ABB RAPID module: Module1.mod

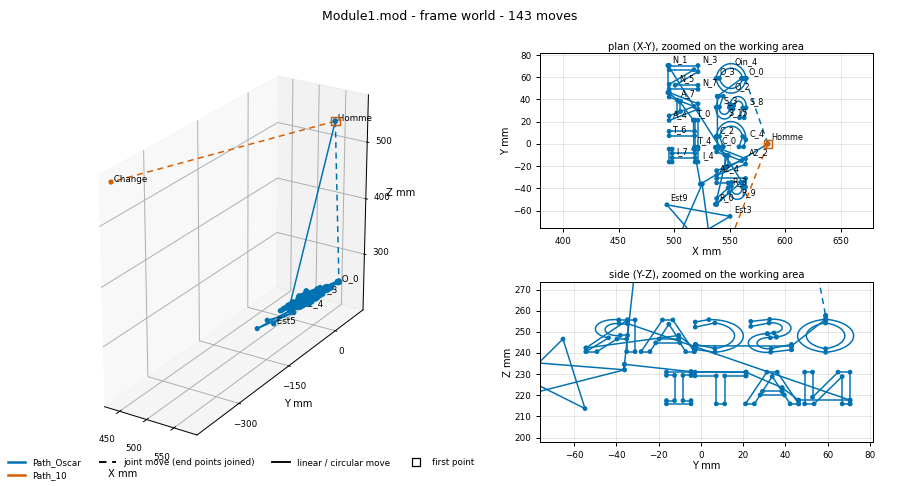
[picture p0: tool path of Module1.mod in frame world, 143 of 143 moves have a stored position in this frame; points joined in program order, loops and branches not executed]
MODULE Module1
    TASK PERS tooldata Marcador:=[TRUE,[[59.777,0,124.777],[0.923879533,0,0.382683432,0]],[0.105,[17.009,0,56.388],[1,0,0,0],0,0,0]];
    TASK PERS wobjdata Pastel:=[FALSE,TRUE,"",[[480,-5.202,208],[0.258819045,0,0.965925826,0]],[[-17.44,75.771,0.905],[0,0,1,0]]];
    CONST robtarget N_1:=[[0,0,2],[0,0,1,0],[-1,1,-2,0],[9E+09,9E+09,9E+09,9E+09,9E+09,9E+09]];
    CONST robtarget N_2:=[[0,0,0],[0,0,1,0],[-1,1,-2,0],[9E+09,9E+09,9E+09,9E+09,9E+09,9E+09]];
    CONST robtarget N_3:=[[30,0,0],[0,0,1,0],[-1,1,-2,0],[9E+09,9E+09,9E+09,9E+09,9E+09,9E+09]];
    CONST robtarget N_4:=[[30,-5.664,0],[0,0,1,0],[-1,1,-2,0],[9E+09,9E+09,9E+09,9E+09,9E+09,9E+09]];
    CONST robtarget N_5:=[[6.248,-17.747,0],[0,0,1,0],[-1,1,-2,0],[9E+09,9E+09,9E+09,9E+09,9E+09,9E+09]];
    CONST robtarget N_6:=[[30,-17.747,0],[0,0,1,0],[-1,1,-2,0],[9E+09,9E+09,9E+09,9E+09,9E+09,9E+09]];
    CONST robtarget N_7:=[[30,-21.467,0],[0,0,1,0],[-1,1,-2,0],[9E+09,9E+09,9E+09,9E+09,9E+09,9E+09]];
    CONST robtarget N_8:=[[-0.000025404,-21.467,0.000044001],[0,0,1,0],[-1,1,-2,0],[9E+09,9E+09,9E+09,9E+09,9E+09,9E+09]];
    CONST robtarget N_9:=[[-0.000025404,-16.993,0.000044001],[0,0,1,0],[-1,1,-2,0],[9E+09,9E+09,9E+09,9E+09,9E+09,9E+09]];
    CONST robtarget N_10:=[[25.867,-3.719,0],[0,0,1,0],[-1,1,-2,0],[9E+09,9E+09,9E+09,9E+09,9E+09,9E+09]];
    CONST robtarget N_11:=[[0,-3.719,0],[0,0,1,0],[-1,1,-2,0],[9E+09,9E+09,9E+09,9E+09,9E+09,9E+09]];
    CONST robtarget N_1_2:=[[0,0,2],[0,0,1,0],[-1,1,-2,0],[9E+09,9E+09,9E+09,9E+09,9E+09,9E+09]];
    CONST robtarget A_0:=[[0,-24.311,2],[0,0,1,0],[-1,1,-2,0],[9E+09,9E+09,9E+09,9E+09,9E+09,9E+09]];
    CONST robtarget A_1:=[[0,-24.311,0],[0,0,1,0],[-1,1,-2,0],[9E+09,9E+09,9E+09,9E+09,9E+09,9E+09]];
    CONST robtarget A_2:=[[30,-34.425,0],[0,0,1,0],[-1,1,-2,0],[9E+09,9E+09,9E+09,9E+09,9E+09,9E+09]];
    CONST robtarget A_3:=[[30,-39.335,0],[0,0,1,0],[-1,1,-2,0],[9E+09,9E+09,9E+09,9E+09,9E+09,9E+09]];
    CONST robtarget A_4:=[[0,-49.449,0],[0,0,1,0],[-1,1,-2,0],[9E+09,9E+09,9E+09,9E+09,9E+09,9E+09]];
    CONST robtarget A_5:=[[0,-45.243,0],[0,0,1,0],[-1,1,-2,0],[9E+09,9E+09,9E+09,9E+09,9E+09,9E+09]];
    CONST robtarget A_6:=[[8.388,-42.52,0],[0,0,1,0],[-1,1,-2,0],[9E+09,9E+09,9E+09,9E+09,9E+09,9E+09]];
    CONST robtarget A_7:=[[8.388,-31.07,0],[0,0,1,0],[-1,1,-2,0],[9E+09,9E+09,9E+09,9E+09,9E+09,9E+09]];
    CONST robtarget A_8:=[[0,-28.347,0],[0,0,1,0],[-1,1,-2,0],[9E+09,9E+09,9E+09,9E+09,9E+09,9E+09]];
    CONST robtarget A_1_2:=[[0,-24.311,0],[0,0,1,0],[-1,1,-2,0],[9E+09,9E+09,9E+09,9E+09,9E+09,9E+09]];
    CONST robtarget A_0_2:=[[0,-24.311,2],[0,0,1,0],[-1,1,-2,0],[9E+09,9E+09,9E+09,9E+09,9E+09,9E+09]];
    CONST robtarget A_in0:=[[11.791,-32.164,2],[0,0,1,0],[-1,1,-2,0],[9E+09,9E+09,9E+09,9E+09,9E+09,9E+09]];
    CONST robtarget A_in1:=[[11.791,-32.164,0],[0,0,1,0],[-1,1,-2,0],[9E+09,9E+09,9E+09,9E+09,9E+09,9E+09]];
    CONST robtarget A_in2:=[[25.916,-36.783,0],[0,0,1,0],[-1,1,-2,0],[9E+09,9E+09,9E+09,9E+09,9E+09,9E+09]];
    CONST robtarget A_in3:=[[11.791,-41.426,0],[0,0,1,0],[-1,1,-2,0],[9E+09,9E+09,9E+09,9E+09,9E+09,9E+09]];
    CONST robtarget A_in1_2:=[[11.791,-32.164,0],[0,0,1,0],[-1,1,-2,0],[9E+09,9E+09,9E+09,9E+09,9E+09,9E+09]];
    CONST robtarget A_in0_2:=[[11.791,-32.164,2],[0,0,1,0],[-1,1,-2,0],[9E+09,9E+09,9E+09,9E+09,9E+09,9E+09]];
    CONST robtarget I_0:=[[26.937,-75.219,2],[0,0,1,0],[-1,1,-2,0],[9E+09,9E+09,9E+09,9E+09,9E+09,9E+09]];
    CONST robtarget I_2:=[[26.937,-75.219,0],[0,0,1,0],[-1,1,-2,0],[9E+09,9E+09,9E+09,9E+09,9E+09,9E+09]];
    CONST robtarget I_3:=[[30,-75.219,0],[0,0,1,0],[-1,1,-2,0],[9E+09,9E+09,9E+09,9E+09,9E+09,9E+09]];
    CONST robtarget I_4:=[[30,-86.839,0],[0,0,1,0],[-1,1,-2,0],[9E+09,9E+09,9E+09,9E+09,9E+09,9E+09]];
    CONST robtarget I_5:=[[26.937,-86.839,0],[0,0,1,0],[-1,1,-2,0],[9E+09,9E+09,9E+09,9E+09,9E+09,9E+09]];
    CONST robtarget I_6:=[[26.937,-83.023,0],[0,0,1,0],[-1,1,-2,0],[9E+09,9E+09,9E+09,9E+09,9E+09,9E+09]];
    CONST robtarget I_7:=[[3.063,-83.023,0],[0,0,1,0],[-1,1,-2,0],[9E+09,9E+09,9E+09,9E+09,9E+09,9E+09]];
    CONST robtarget I_8:=[[3.063,-86.839,0],[0,0,1,0],[-1,1,-2,0],[9E+09,9E+09,9E+09,9E+09,9E+09,9E+09]];
    CONST robtarget I_9:=[[0,-86.839,0],[0,0,1,0],[-1,1,-2,0],[9E+09,9E+09,9E+09,9E+09,9E+09,9E+09]];
    CONST robtarget I_10:=[[0,-75.219,0],[0,0,1,0],[-1,1,-2,0],[9E+09,9E+09,9E+09,9E+09,9E+09,9E+09]];
    CONST robtarget I_11:=[[3.063,-75.219,0],[0,0,1,0],[-1,1,-2,0],[9E+09,9E+09,9E+09,9E+09,9E+09,9E+09]];
    CONST robtarget I_12:=[[3.063,-79.036,0],[0,0,1,0],[-1,1,-2,0],[9E+09,9E+09,9E+09,9E+09,9E+09,9E+09]];
    CONST robtarget I_13:=[[26.937,-79.036,0],[0,0,1,0],[-1,1,-2,0],[9E+09,9E+09,9E+09,9E+09,9E+09,9E+09]];
    CONST robtarget I_2_2:=[[26.937,-75.219,0],[0,0,1,0],[-1,1,-2,0],[9E+09,9E+09,9E+09,9E+09,9E+09,9E+09]];
    CONST robtarget I_0_2:=[[26.937,-75.219,2],[0,0,1,0],[-1,1,-2,0],[9E+09,9E+09,9E+09,9E+09,9E+09,9E+09]];
    CONST robtarget T_0:=[[26.451,-49.23,2],[0,0,1,0],[-1,1,-2,0],[9E+09,9E+09,9E+09,9E+09,9E+09,9E+09]];
    CONST robtarget T_1:=[[26.451,-49.23,0],[0,0,1,0],[-1,1,-2,0],[9E+09,9E+09,9E+09,9E+09,9E+09,9E+09]];
    CONST robtarget T_2:=[[30,-49.23,0],[0,0,1,0],[-1,1,-2,0],[9E+09,9E+09,9E+09,9E+09,9E+09,9E+09]];
    CONST robtarget T_3:=[[30,-73.347,0],[0,0,1,0],[-1,1,-2,0],[9E+09,9E+09,9E+09,9E+09,9E+09,9E+09]];
    CONST robtarget T_4:=[[26.451,-73.347,0],[0,0,1,0],[-1,1,-2,0],[9E+09,9E+09,9E+09,9E+09,9E+09,9E+09]];
    CONST robtarget T_5:=[[26.451,-63.282,0],[0,0,1,0],[-1,1,-2,0],[9E+09,9E+09,9E+09,9E+09,9E+09,9E+09]];
    CONST robtarget T_6:=[[0,-63.282,0],[0,0,1,0],[-1,1,-2,0],[9E+09,9E+09,9E+09,9E+09,9E+09,9E+09]];
    CONST robtarget T_7:=[[0,-59.295,0],[0,0,1,0],[-1,1,-2,0],[9E+09,9E+09,9E+09,9E+09,9E+09,9E+09]];
    CONST robtarget T_8:=[[26.451,-59.295,0],[0,0,1,0],[-1,1,-2,0],[9E+09,9E+09,9E+09,9E+09,9E+09,9E+09]];
    CONST robtarget T_1_2:=[[26.451,-49.23,0],[0,0,1,0],[-1,1,-2,0],[9E+09,9E+09,9E+09,9E+09,9E+09,9E+09]];
    CONST robtarget T_0_2:=[[26.451,-49.23,2],[0,0,1,0],[-1,1,-2,0],[9E+09,9E+09,9E+09,9E+09,9E+09,9E+09]];
    CONST robtarget A2_0:=[[49.394,-73.711,2],[0,0,1,0],[-1,1,-2,0],[9E+09,9E+09,9E+09,9E+09,9E+09,9E+09]];
    CONST robtarget A2_1:=[[49.394,-73.711,0],[0,0,1,0],[-1,1,-2,0],[9E+09,9E+09,9E+09,9E+09,9E+09,9E+09]];
    CONST robtarget A2_2:=[[79.394,-83.825,0],[0,0,1,0],[-1,1,-2,0],[9E+09,9E+09,9E+09,9E+09,9E+09,9E+09]];
    CONST robtarget A2_3:=[[79.394,-88.736,0],[0,0,1,0],[-1,1,-2,0],[9E+09,9E+09,9E+09,9E+09,9E+09,9E+09]];
    CONST robtarget A2_4:=[[49.394,-98.849,0],[0,0,1,0],[-1,1,-2,0],[9E+09,9E+09,9E+09,9E+09,9E+09,9E+09]];
    CONST robtarget A2_5:=[[49.394,-94.643,0],[0,0,1,0],[-1,1,-2,0],[9E+09,9E+09,9E+09,9E+09,9E+09,9E+09]];
    CONST robtarget A2_6:=[[57.782,-91.92,0],[0,0,1,0],[-1,1,-2,0],[9E+09,9E+09,9E+09,9E+09,9E+09,9E+09]];
    CONST robtarget A2_7:=[[57.782,-80.47,0],[0,0,1,0],[-1,1,-2,0],[9E+09,9E+09,9E+09,9E+09,9E+09,9E+09]];
    CONST robtarget A2_8:=[[49.394,-77.747,0],[0,0,1,0],[-1,1,-2,0],[9E+09,9E+09,9E+09,9E+09,9E+09,9E+09]];
    CONST robtarget A2_1_2:=[[49.394,-73.711,0],[0,0,1,0],[-1,1,-2,0],[9E+09,9E+09,9E+09,9E+09,9E+09,9E+09]];
    CONST robtarget A2_0_2:=[[49.394,-73.711,2],[0,0,1,0],[-1,1,-2,0],[9E+09,9E+09,9E+09,9E+09,9E+09,9E+09]];
    CONST robtarget C_0:=[[51.437,-73.225,2],[0,0,1,0],[-1,1,-2,0],[9E+09,9E+09,9E+09,9E+09,9E+09,9E+09]];
    CONST robtarget C_1:=[[51.437,-73.225,0],[0,0,1,0],[-1,1,-2,0],[9E+09,9E+09,9E+09,9E+09,9E+09,9E+09]];
    CONST robtarget C_2:=[[48.86,-63.89,0],[0,0,1,0],[-1,1,-2,0],[9E+09,9E+09,9E+09,9E+09,9E+09,9E+09]];
    CONST robtarget C_3:=[[64.37,-50.47,0],[0,0,1,0],[-1,1,-2,0],[9E+09,9E+09,9E+09,9E+09,9E+09,9E+09]];
    CONST robtarget C_4:=[[79.71,-66.795,0],[0,0,1,0],[-1,1,-2,0],[9E+09,9E+09,9E+09,9E+09,9E+09,9E+09]];
    CONST robtarget C_5:=[[77.401,-73.225,0],[0,0,1,0],[-1,1,-2,0],[9E+09,9E+09,9E+09,9E+09,9E+09,9E+09]];
    CONST robtarget C_6:=[[72.587,-73.225,0],[0,0,1,0],[-1,1,-2,0],[9E+09,9E+09,9E+09,9E+09,9E+09,9E+09]];
    CONST robtarget C_7:=[[76.526,-63.938,0],[0,0,1,0],[-1,1,-2,0],[9E+09,9E+09,9E+09,9E+09,9E+09,9E+09]];
    CONST robtarget C_8:=[[64.37,-54.627,0],[0,0,1,0],[-1,1,-2,0],[9E+09,9E+09,9E+09,9E+09,9E+09,9E+09]];
    CONST robtarget C_9:=[[52.312,-63.938,0],[0,0,1,0],[-1,1,-2,0],[9E+09,9E+09,9E+09,9E+09,9E+09,9E+09]];
    CONST robtarget C_10:=[[56.202,-72.933,0],[0,0,1,0],[-1,1,-2,0],[9E+09,9E+09,9E+09,9E+09,9E+09,9E+09]];
    CONST robtarget C_11:=[[56.202,-73.225,0],[0,0,1,0],[-1,1,-2,0],[9E+09,9E+09,9E+09,9E+09,9E+09,9E+09]];
    CONST robtarget C_1_2:=[[51.437,-73.225,0],[0,0,1,0],[-1,1,-2,0],[9E+09,9E+09,9E+09,9E+09,9E+09,9E+09]];
    CONST robtarget S_0:=[[51.193,-27.715,2],[0,0,1,0],[-1,1,-2,0],[9E+09,9E+09,9E+09,9E+09,9E+09,9E+09]];
    CONST robtarget S_1:=[[51.193,-27.715,0],[0,0,1,0],[-1,1,-2,0],[9E+09,9E+09,9E+09,9E+09,9E+09,9E+09]];
    CONST robtarget S_2:=[[56.202,-27.715,0],[0,0,1,0],[-1,1,-2,0],[9E+09,9E+09,9E+09,9E+09,9E+09,9E+09]];
    CONST robtarget S_3:=[[52.312,-37.269,0],[0,0,1,0],[-1,1,-2,0],[9E+09,9E+09,9E+09,9E+09,9E+09,9E+09]];
    CONST robtarget S_4:=[[57.32,-43.954,0],[0,0,1,0],[-1,1,-2,0],[9E+09,9E+09,9E+09,9E+09,9E+09,9E+09]];
    CONST robtarget S_Mid:=[[62.570793399,-37.719,-0.000172845],[0,0,1,0],[-1,1,-2,0],[9E+09,9E+09,9E+09,9E+09,9E+09,9E+09]];
    CONST robtarget S_5:=[[63.276,-34.838,0],[0,0,1,0],[-1,1,-2,0],[9E+09,9E+09,9E+09,9E+09,9E+09,9E+09]];
    CONST robtarget S_6:=[[63.276,-34.838,0],[0,0,1,0],[-1,1,-2,0],[9E+09,9E+09,9E+09,9E+09,9E+09,9E+09]];
    CONST robtarget S_7:=[[71.347,-27.933,0],[0,0,1,0],[-1,1,-2,0],[9E+09,9E+09,9E+09,9E+09,9E+09,9E+09]];
    CONST robtarget S_8:=[[79.929,-38.023,0],[0,0,1,0],[-1,1,-2,0],[9E+09,9E+09,9E+09,9E+09,9E+09,9E+09]];
    CONST robtarget S_9:=[[77.984,-46.945,0],[0,0,1,0],[-1,1,-2,0],[9E+09,9E+09,9E+09,9E+09,9E+09,9E+09]];
    CONST robtarget S_10:=[[73.219,-46.945,0],[0,0,1,0],[-1,1,-2,0],[9E+09,9E+09,9E+09,9E+09,9E+09,9E+09]];
    CONST robtarget S_11:=[[76.477,-38.29,0],[0,0,1,0],[-1,1,-2,0],[9E+09,9E+09,9E+09,9E+09,9E+09,9E+09]];
    CONST robtarget S_12:=[[71.761,-32.091,0],[0,0,1,0],[-1,1,-2,0],[9E+09,9E+09,9E+09,9E+09,9E+09,9E+09]];
    CONST robtarget S_Mid2:=[[67.09264888,-36.005,-0.000089407],[0,0,1,0],[-1,1,-2,0],[9E+09,9E+09,9E+09,9E+09,9E+09,9E+09]];
    CONST robtarget S_13:=[[66.315,-39.104,0],[0,0,1,0],[-1,1,-2,0],[9E+09,9E+09,9E+09,9E+09,9E+09,9E+09]];
    CONST robtarget S_14:=[[66.315,-39.104,0],[0,0,1,0],[-1,1,-2,0],[9E+09,9E+09,9E+09,9E+09,9E+09,9E+09]];
    CONST robtarget S_15:=[[57.952,-48.112,0],[0,0,1,0],[-1,1,-2,0],[9E+09,9E+09,9E+09,9E+09,9E+09,9E+09]];
    CONST robtarget S_16:=[[48.86,-37.561,0],[0,0,1,0],[-1,1,-2,0],[9E+09,9E+09,9E+09,9E+09,9E+09,9E+09]];
    CONST robtarget Homme:=[[251.699224046,-70.569,258.141906106],[0.130526192,0,-0.991444861,0],[-1,1,-2,0],[9E+09,9E+09,9E+09,9E+09,9E+09,9E+09]];
    CONST robtarget O_0:=[[80.026,-11.548,2],[0,0,1,0],[-1,1,-2,0],[9E+09,9E+09,9E+09,9E+09,9E+09,9E+09]];
    CONST robtarget O_1:=[[80.026,-11.548,0],[0,0,1,0],[-1,1,-2,0],[9E+09,9E+09,9E+09,9E+09,9E+09,9E+09]];
    CONST robtarget O_2:=[[64.394,-24.822,0],[0,0,1,0],[-1,1,-2,0],[9E+09,9E+09,9E+09,9E+09,9E+09,9E+09]];
    CONST robtarget O_3:=[[48.762,-11.548,0],[0,0,1,0],[-1,1,-2,0],[9E+09,9E+09,9E+09,9E+09,9E+09,9E+09]];
    CONST robtarget O_4:=[[64.394,1.702,0],[0,0,1,0],[-1,1,-2,0],[9E+09,9E+09,9E+09,9E+09,9E+09,9E+09]];
    CONST robtarget Oin_0:=[[76.574,-11.572,2],[0,0,1,0],[-1,1,-2,0],[9E+09,9E+09,9E+09,9E+09,9E+09,9E+09]];
    CONST robtarget Oin_1:=[[76.574,-11.572,0],[0,0,1,0],[-1,1,-2,0],[9E+09,9E+09,9E+09,9E+09,9E+09,9E+09]];
    CONST robtarget Oin_2:=[[64.394,-20.664,0],[0,0,1,0],[-1,1,-2,0],[9E+09,9E+09,9E+09,9E+09,9E+09,9E+09]];
    CONST robtarget Oin_3:=[[52.214,-11.572,0],[0,0,1,0],[-1,1,-2,0],[9E+09,9E+09,9E+09,9E+09,9E+09,9E+09]];
    CONST robtarget Oin_4:=[[64.394,-2.455,0],[0,0,1,0],[-1,1,-2,0],[9E+09,9E+09,9E+09,9E+09,9E+09,9E+09]];
    CONST robtarget R_0:=[[49.394,-124.911,2],[0,0,1,0],[-1,1,-2,0],[9E+09,9E+09,9E+09,9E+09,9E+09,9E+09]];
    CONST robtarget R_1:=[[49.394,-124.911,0],[0,0,1,0],[-1,1,-2,0],[9E+09,9E+09,9E+09,9E+09,9E+09,9E+09]];
    CONST robtarget R_2:=[[49.394,-119.732,0],[0,0,1,0],[-1,1,-2,0],[9E+09,9E+09,9E+09,9E+09,9E+09,9E+09]];
    CONST robtarget R_3:=[[61.331,-110.251,0],[0,0,1,0],[-1,1,-2,0],[9E+09,9E+09,9E+09,9E+09,9E+09,9E+09]];
    CONST robtarget R_4:=[[61.331,-105.681,0],[0,0,1,0],[-1,1,-2,0],[9E+09,9E+09,9E+09,9E+09,9E+09,9E+09]];
    CONST robtarget R_5:=[[49.394,-105.681,0],[0,0,1,0],[-1,1,-2,0],[9E+09,9E+09,9E+09,9E+09,9E+09,9E+09]];
    CONST robtarget R_6:=[[49.394,-101.694,0],[0,0,1,0],[-1,1,-2,0],[9E+09,9E+09,9E+09,9E+09,9E+09,9E+09]];
    CONST robtarget R_7:=[[79.394,-101.694,0],[0,0,1,0],[-1,1,-2,0],[9E+09,9E+09,9E+09,9E+09,9E+09,9E+09]];
    CONST robtarget R_8:=[[79.394,-109.425,0],[0,0,1,0],[-1,1,-2,0],[9E+09,9E+09,9E+09,9E+09,9E+09,9E+09]];
    CONST robtarget R_9:=[[71.25,-120.462,0],[0,0,1,0],[-1,1,-2,0],[9E+09,9E+09,9E+09,9E+09,9E+09,9E+09]];
    CONST robtarget R_10:=[[62.449,-114.238,0],[0,0,1,0],[-1,1,-2,0],[9E+09,9E+09,9E+09,9E+09,9E+09,9E+09]];
    CONST robtarget A2in_0:=[[61.224,-81.097,2],[0,0,1,0],[-1,1,-2,0],[9E+09,9E+09,9E+09,9E+09,9E+09,9E+09]];
    CONST robtarget A2in_1:=[[61.224,-81.097,0],[0,0,1,0],[-1,1,-2,0],[9E+09,9E+09,9E+09,9E+09,9E+09,9E+09]];
    CONST robtarget A2in_2:=[[75.349,-85.716,0],[0,0,1,0],[-1,1,-2,0],[9E+09,9E+09,9E+09,9E+09,9E+09,9E+09]];
    CONST robtarget A2in_3:=[[61.224,-90.36,0],[0,0,1,0],[-1,1,-2,0],[9E+09,9E+09,9E+09,9E+09,9E+09,9E+09]];
    CONST robtarget Rin_0:=[[75.981,-105.214,2],[0,0,1,0],[-1,1,-2,0],[9E+09,9E+09,9E+09,9E+09,9E+09,9E+09]];
    CONST robtarget Rin_1:=[[75.981,-105.214,0],[0,0,1,0],[-1,1,-2,0],[9E+09,9E+09,9E+09,9E+09,9E+09,9E+09]];
    CONST robtarget Rin_2:=[[75.981,-109.177,0],[0,0,1,0],[-1,1,-2,0],[9E+09,9E+09,9E+09,9E+09,9E+09,9E+09]];
    CONST robtarget Rin_3:=[[70.973,-115.838,0],[0,0,1,0],[-1,1,-2,0],[9E+09,9E+09,9E+09,9E+09,9E+09,9E+09]];
    CONST robtarget Rin_4:=[[64.701,-108.715,0],[0,0,1,0],[-1,1,-2,0],[9E+09,9E+09,9E+09,9E+09,9E+09,9E+09]];
    CONST robtarget Rin_5:=[[64.701,-105.214,0],[0,0,1,0],[-1,1,-2,0],[9E+09,9E+09,9E+09,9E+09,9E+09,9E+09]];
    CONST robtarget Est4:=[[15.21,-147.353,-0.905],[0.021468987,0,-0.999769515,0],[-1,1,-2,0],[9E+09,9E+09,9E+09,9E+09,9E+09,9E+09]];
    CONST robtarget Est5:=[[44.188,-172.469,-0.905],[0,0,1,0],[-1,1,-2,0],[9E+09,9E+09,9E+09,9E+09,9E+09,9E+09]];
    CONST robtarget Est6:=[[1.207,-154.488,-0.905],[0.015437258,0,-0.999880838,0],[-1,1,-2,0],[9E+09,9E+09,9E+09,9E+09,9E+09,9E+09]];
    CONST robtarget Est7:=[[3.549,-166.033,-0.905],[0,0,1,0],[-1,1,-2,0],[9E+09,9E+09,9E+09,9E+09,9E+09,9E+09]];
    CONST robtarget Est8:=[[-9.906,-143.375,-0.905],[0.009404795,0,-0.999955774,0],[-1,1,-2,0],[9E+09,9E+09,9E+09,9E+09,9E+09,9E+09]];
    CONST robtarget Est10:=[[-2.771,-129.372,-0.905],[0.003372162,0,-0.999994314,0],[-1,1,-2,0],[9E+09,9E+09,9E+09,9E+09,9E+09,9E+09]];
    CONST robtarget Est0_2:=[[33.773,-106.715,2.095],[0,0,1,0],[-1,1,-2,0],[9E+09,9E+09,9E+09,9E+09,9E+09,9E+09]];
    CONST robtarget Est0:=[[33.773,-106.715,2.095],[0,0,1,0],[-1,1,-2,0],[9E+09,9E+09,9E+09,9E+09,9E+09,9E+09]];
    CONST robtarget Est1:=[[33.773,-106.715,-0.905],[0,0,1,0],[-1,1,-2,0],[9E+09,9E+09,9E+09,9E+09,9E+09,9E+09]];
    CONST robtarget Est1_2:=[[33.773,-106.715,-0.905],[0,0,1,0],[-1,1,-2,0],[9E+09,9E+09,9E+09,9E+09,9E+09,9E+09]];
    CONST robtarget Est3:=[[62.867,-135.809,-0.905],[0,0,1,0],[-1,1,-2,0],[9E+09,9E+09,9E+09,9E+09,9E+09,9E+09]];
    CONST robtarget Est2:=[[12.751,-131.831,-0.905],[0.027499868,0,-0.999621807,0],[-1,1,-2,0],[9E+09,9E+09,9E+09,9E+09,9E+09,9E+09]];
    CONST robtarget Est9:=[[-2.887,-125.394,-0.905],[0,0,1,0],[-1,1,-2,0],[9E+09,9E+09,9E+09,9E+09,9E+09,9E+09]];
    CONST robtarget Change:=[[117.149200276,-467.39587511,335.823939412],[0.121542778,-0.336820162,-0.923209057,0.13951548],[-1,1,-2,0],[9E+09,9E+09,9E+09,9E+09,9E+09,9E+09]];

    PROC main()
        WaitDI Trayectoria,1;
        Path_Oscar;
        WaitDI Mantenimiento,1;
        Path_10;
    ENDPROC
    PROC Path_Oscar()
        MoveL Homme,v100,fine,Marcador\WObj:=Pastel;
        MoveJ O_0,v100,z100,Marcador\WObj:=Pastel;
        MoveL O_1,v100,z100,Marcador\WObj:=Pastel;
        MoveC O_2,O_3,v100,z100,Marcador\WObj:=Pastel;
        MoveC O_4,O_1,v100,z100,Marcador\WObj:=Pastel;
        MoveL O_0,v100,z100,Marcador\WObj:=Pastel;
        MoveL Oin_0,v100,z100,Marcador\WObj:=Pastel;
        MoveL Oin_1,v100,z100,Marcador\WObj:=Pastel;
        MoveC Oin_2,Oin_3,v100,z100,Marcador\WObj:=Pastel;
        MoveC Oin_4,Oin_1,v100,z100,Marcador\WObj:=Pastel;
        MoveL Oin_0,v100,z100,Marcador\WObj:=Pastel;
        MoveL S_0,v100,z100,Marcador\WObj:=Pastel;
        MoveL S_1,v100,z100,Marcador\WObj:=Pastel;
        MoveL S_2,v100,z100,Marcador\WObj:=Pastel;
        MoveL S_3,v100,z100,Marcador\WObj:=Pastel;
        MoveC S_4,S_Mid,v100,z100,Marcador\WObj:=Pastel;
        MoveL S_5,v100,z100,Marcador\WObj:=Pastel;
        MoveL S_6,v100,z100,Marcador\WObj:=Pastel;
        MoveC S_7,S_8,v100,z100,Marcador\WObj:=Pastel;
        MoveL S_9,v100,z100,Marcador\WObj:=Pastel;
        MoveL S_10,v100,z100,Marcador\WObj:=Pastel;
        MoveL S_11,v100,z100,Marcador\WObj:=Pastel;
        MoveC S_12,S_Mid2,v100,z100,Marcador\WObj:=Pastel;
        MoveL S_13,v100,z100,Marcador\WObj:=Pastel;
        MoveL S_14,v100,z100,Marcador\WObj:=Pastel;
        MoveC S_15,S_16,v100,z100,Marcador\WObj:=Pastel;
        MoveL S_1,v100,z100,Marcador\WObj:=Pastel;
        MoveL S_0,v100,z100,Marcador\WObj:=Pastel;
        MoveL C_0,v100,z100,Marcador\WObj:=Pastel;
        MoveL C_1,v100,z100,Marcador\WObj:=Pastel;
        MoveL C_2,v100,z100,Marcador\WObj:=Pastel;
        MoveC C_3,C_4,v100,z100,Marcador\WObj:=Pastel;
        MoveL C_5,v100,z100,Marcador\WObj:=Pastel;
        MoveL C_6,v100,z100,Marcador\WObj:=Pastel;
        MoveL C_7,v100,z100,Marcador\WObj:=Pastel;
        MoveC C_8,C_9,v100,z100,Marcador\WObj:=Pastel;
        MoveL C_10,v100,z100,Marcador\WObj:=Pastel;
        MoveL C_11,v100,z100,Marcador\WObj:=Pastel;
        MoveL C_1_2,v100,z100,Marcador\WObj:=Pastel;
        MoveL C_0,v100,z100,Marcador\WObj:=Pastel;
        MoveL A2_0,v100,z100,Marcador\WObj:=Pastel;
        MoveL A2_1,v100,z100,Marcador\WObj:=Pastel;
        MoveL A2_2,v100,z100,Marcador\WObj:=Pastel;
        MoveL A2_3,v100,z100,Marcador\WObj:=Pastel;
        MoveL A2_4,v100,z100,Marcador\WObj:=Pastel;
        MoveL A2_5,v100,z100,Marcador\WObj:=Pastel;
        MoveL A2_6,v100,z100,Marcador\WObj:=Pastel;
        MoveL A2_7,v100,z100,Marcador\WObj:=Pastel;
        MoveL A2_8,v100,z100,Marcador\WObj:=Pastel;
        MoveL A2_1_2,v100,z100,Marcador\WObj:=Pastel;
        MoveL A2_0_2,v100,z100,Marcador\WObj:=Pastel;
        MoveL A2in_0,v100,z100,Marcador\WObj:=Pastel;
        MoveL A2in_1,v100,z100,Marcador\WObj:=Pastel;
        MoveL A2in_2,v100,z100,Marcador\WObj:=Pastel;
        MoveL A2in_3,v100,z100,Marcador\WObj:=Pastel;
        MoveL A2in_1,v100,z100,Marcador\WObj:=Pastel;
        MoveL A2in_0,v100,z100,Marcador\WObj:=Pastel;
        MoveL R_0,v100,z100,Marcador\WObj:=Pastel;
        MoveL R_1,v100,z100,Marcador\WObj:=Pastel;
        MoveL R_2,v100,z100,Marcador\WObj:=Pastel;
        MoveL R_3,v100,z100,Marcador\WObj:=Pastel;
        MoveL R_4,v100,z100,Marcador\WObj:=Pastel;
        MoveL R_5,v100,z100,Marcador\WObj:=Pastel;
        MoveL R_6,v100,z100,Marcador\WObj:=Pastel;
        MoveL R_7,v100,z100,Marcador\WObj:=Pastel;
        MoveL R_8,v100,z100,Marcador\WObj:=Pastel;
        MoveC R_9,R_10,v100,z100,Marcador\WObj:=Pastel;
        MoveL R_1,v100,z100,Marcador\WObj:=Pastel;
        MoveL R_0,v100,z100,Marcador\WObj:=Pastel;
        MoveL Rin_0,v100,z100,Marcador\WObj:=Pastel;
        MoveL Rin_1,v100,z100,Marcador\WObj:=Pastel;
        MoveL Rin_2,v100,z100,Marcador\WObj:=Pastel;
        MoveC Rin_3,Rin_4,v100,z100,Marcador\WObj:=Pastel;
        MoveL Rin_5,v100,z100,Marcador\WObj:=Pastel;
        MoveL Rin_0,v100,z100,Marcador\WObj:=Pastel;
        MoveL Rin_1,v100,z100,Marcador\WObj:=Pastel;
        MoveL N_1,v200,fine,Marcador\WObj:=Pastel;
        MoveL N_2,v200,fine,Marcador\WObj:=Pastel;
        MoveL N_3,v200,fine,Marcador\WObj:=Pastel;
        MoveL N_4,v200,fine,Marcador\WObj:=Pastel;
        MoveL N_5,v200,fine,Marcador\WObj:=Pastel;
        MoveL N_6,v200,fine,Marcador\WObj:=Pastel;
        MoveL N_7,v200,fine,Marcador\WObj:=Pastel;
        MoveL N_8,v200,fine,Marcador\WObj:=Pastel;
        MoveL N_9,v200,fine,Marcador\WObj:=Pastel;
        MoveL N_10,v200,fine,Marcador\WObj:=Pastel;
        MoveL N_11,v200,fine,Marcador\WObj:=Pastel;
        MoveL N_2,v200,fine,Marcador\WObj:=Pastel;
        MoveL N_1_2,v200,fine,Marcador\WObj:=Pastel;
        MoveL A_0,v100,z100,Marcador\WObj:=Pastel;
        MoveL A_1,v100,z100,Marcador\WObj:=Pastel;
        MoveL A_2,v100,z100,Marcador\WObj:=Pastel;
        MoveL A_3,v100,z100,Marcador\WObj:=Pastel;
        MoveL A_4,v100,z100,Marcador\WObj:=Pastel;
        MoveL A_5,v100,z100,Marcador\WObj:=Pastel;
        MoveL A_6,v100,z100,Marcador\WObj:=Pastel;
        MoveL A_7,v100,z100,Marcador\WObj:=Pastel;
        MoveL A_8,v100,z100,Marcador\WObj:=Pastel;
        MoveL A_1_2,v100,z100,Marcador\WObj:=Pastel;
        MoveL A_0_2,v100,z100,Marcador\WObj:=Pastel;
        MoveL A_in0,v100,z100,Marcador\WObj:=Pastel;
        MoveL A_in1,v100,z100,Marcador\WObj:=Pastel;
        MoveL A_in2,v100,z100,Marcador\WObj:=Pastel;
        MoveL A_in3,v100,z100,Marcador\WObj:=Pastel;
        MoveL A_in1,v100,z100,Marcador\WObj:=Pastel;
        MoveL A_in0,v100,z100,Marcador\WObj:=Pastel;
        MoveL T_0,v100,z100,Marcador\WObj:=Pastel;
        MoveL T_1,v100,z100,Marcador\WObj:=Pastel;
        MoveL T_2,v100,z100,Marcador\WObj:=Pastel;
        MoveL T_3,v100,z100,Marcador\WObj:=Pastel;
        MoveL T_4,v100,z100,Marcador\WObj:=Pastel;
        MoveL T_5,v100,z100,Marcador\WObj:=Pastel;
        MoveL T_6,v100,z100,Marcador\WObj:=Pastel;
        MoveL T_7,v100,z100,Marcador\WObj:=Pastel;
        MoveL T_8,v100,z100,Marcador\WObj:=Pastel;
        MoveL T_1_2,v100,z100,Marcador\WObj:=Pastel;
        MoveL T_0_2,v100,z100,Marcador\WObj:=Pastel;
        MoveL I_0,v100,z100,Marcador\WObj:=Pastel;
        MoveL I_2,v100,z100,Marcador\WObj:=Pastel;
        MoveL I_3,v100,z100,Marcador\WObj:=Pastel;
        MoveL I_4,v100,z100,Marcador\WObj:=Pastel;
        MoveL I_5,v100,z100,Marcador\WObj:=Pastel;
        MoveL I_6,v100,z100,Marcador\WObj:=Pastel;
        MoveL I_7,v100,z100,Marcador\WObj:=Pastel;
        MoveL I_8,v100,z100,Marcador\WObj:=Pastel;
        MoveL I_9,v100,z100,Marcador\WObj:=Pastel;
        MoveL I_10,v100,z100,Marcador\WObj:=Pastel;
        MoveL I_11,v100,z100,Marcador\WObj:=Pastel;
        MoveL I_12,v100,z100,Marcador\WObj:=Pastel;
        MoveL I_13,v100,z100,Marcador\WObj:=Pastel;
        MoveL I_2_2,v100,z100,Marcador\WObj:=Pastel;
        MoveL I_0_2,v100,z100,Marcador\WObj:=Pastel;
        MoveL Est0,v100,z100,Marcador\WObj:=Pastel;
        MoveL Est1,v100,fine,Marcador\WObj:=Pastel;
        MoveL Est5,v100,fine,Marcador\WObj:=Pastel;
        MoveL Est9,v100,fine,Marcador\WObj:=Pastel;
        MoveL Est3,v100,fine,Marcador\WObj:=Pastel;
        MoveL Est7,v100,fine,Marcador\WObj:=Pastel;
        MoveL Est1_2,v100,fine,Marcador\WObj:=Pastel;
        MoveL Est0_2,v100,fine,Marcador\WObj:=Pastel;
        MoveL Homme,v100,fine,Marcador\WObj:=Pastel;
    ENDPROC
    PROC Path_10()
        MoveL Homme,v100,fine,Marcador\WObj:=Pastel;
        MoveJ Change,v100,z100,Marcador\WObj:=Pastel;
    ENDPROC
ENDMODULE
